Yaskawa INFORM job: X2_NOWY2.JBI

/JOB
//NAME X2_NOWY2
//POS
///NPOS 322,322,322,20,0,0
///TOOL 0
///POSTYPE PULSE
///PULSE
C00000=1579,-114561,-88072,141,60969,-160
C00001=1579,-126069,-115869,130,72161,-147
C00002=-67532,-124352,-115339,134,72718,-152
C00003=-81630,-76415,-67707,7081,99866,-75616
C00004=-81630,-76414,-67706,7081,99866,-75616
C00005=-85213,-86895,-71424,6566,97096,-77009
C00006=-85213,-86471,-70205,6561,96571,-77039
C00007=-85213,-86895,-71424,6566,97096,-77009
C00008=-86383,-83236,-69405,6430,97828,-77376
C00009=-86383,-82993,-68650,6424,97491,-77394
C00010=-85656,-85286,-69628,6508,96860,-77177
C00011=-86054,-83030,-69774,6481,98134,-77248
C00012=-91609,-64546,-67425,5952,106567,-78770
C00013=-108338,-72557,-69392,19017,102016,-84323
C00014=-103994,-87799,-70649,19047,94316,-83966
C00015=-101914,-94753,-72721,19202,91650,-83636
C00016=-101720,-95093,-71454,19192,90702,-83718
C00017=-101720,-95403,-72147,19196,90955,-83679
C00018=-102509,-90897,-70406,19144,92318,-83747
C00019=-102509,-90529,-69509,19136,91974,-83801
C00020=-102070,-93055,-70499,19166,91217,-83763
C00021=-103193,-87364,-70534,19135,94271,-83684
C00022=-105000,-74500,-64879,19101,97659,-83800
C00023=-113069,-60767,-53247,26239,106025,-84622
C00024=-112828,-63942,-52646,27281,108527,-83919
C00025=-112433,-69525,-54608,27546,108328,-83811
C00026=-112433,-69174,-53580,27467,107925,-83912
C00027=-112433,-68598,-51946,27347,107292,-84070
C00028=-112433,-68839,-52622,27396,107553,-84005
C00029=-112673,-65386,-50917,27452,108279,-83921
C00030=-112744,-64051,-49536,27403,108156,-83979
C00031=-112560,-66748,-50889,27360,107600,-84043
C00032=-112776,-63836,-50109,27476,108578,-83887
C00033=-126682,-57830,-51235,23795,116313,-87772
C00034=-91609,-64546,-67425,5952,106567,-78770
C00035=-73590,-134956,-134527,8565,110042,-72105
C00036=-73590,-134956,-134527,8565,110042,-72105
C00037=-85079,-90579,-82104,6699,101738,-76716
C00038=-105233,-99145,-78854,31145,91869,-85162
C00039=-91621,-98116,-75011,30201,81397,-82609
C00040=-84913,-93599,-68771,30087,77670,-80961
C00041=-84913,-92982,-67436,30137,77231,-81076
C00042=-84913,-93205,-67917,30119,77389,-81035
C00043=-86149,-89803,-66593,30086,78643,-81188
C00044=-86149,-89533,-65979,30106,78434,-81245
C00045=-85360,-91719,-66835,30129,77634,-81148
C00046=-89786,-90500,-68269,30172,80536,-82119
C00047=-91499,-86657,-71640,30020,84676,-81700
C00048=-78974,-84836,-79700,7511,102662,-74517
C00049=-79298,-82189,-71657,7361,99132,-74844
C00050=-79260,-81836,-70076,7347,98342,-74878
C00051=-79260,-81218,-68032,7328,97407,-74935
C00052=-79260,-81362,-68495,7333,97617,-74923
C00053=-80441,-78182,-67079,7204,98482,-75282
C00054=-80441,-78012,-66485,7183,98203,-75298
C00055=-79756,-79865,-67316,7258,97705,-75089
C00056=-80252,-78819,-67734,7202,98493,-75213
C00057=-80252,-80316,-73749,7282,101403,-75042
C00058=-98731,-93358,-79222,4709,99471,-81580
C00059=-98353,-93948,-76089,4728,97224,-81535
C00060=-98128,-94312,-74616,4747,96121,-81500
C00061=-98128,-93684,-73071,4742,95494,-81523
C00062=-98128,-93884,-73558,4744,95690,-81516
C00063=-98894,-90114,-72074,4647,96754,-81739
C00064=-98894,-89854,-71388,4644,96467,-81750
C00065=-98435,-92128,-72291,4703,95830,-81616
C00066=-99279,-88707,-72907,4606,98011,-81825
C00067=-99279,-90964,-80150,4662,101298,-81702
C00068=-83031,-73882,-65637,-17912,114082,-77307
C00069=-85653,-78852,-59840,-26006,111225,-77738
C00070=-86395,-77948,-56111,-25174,109013,-77551
C00071=-86395,-77463,-54950,-25096,108589,-77455
C00072=-86395,-77605,-55287,-25118,108711,-77483
C00073=-87408,-74561,-53917,-25584,109056,-77966
C00074=-87408,-74338,-53367,-25545,108852,-77918
C00075=-86830,-76093,-54163,-25280,108655,-77643
C00076=-86155,-69275,-53538,-25095,111477,-78039
C00077=-82305,-66217,-52035,-23871,113209,-76862
C00078=-98731,-93358,-79222,4709,99471,-81580
C00079=-87850,-130184,-128808,6122,98008,-77863
C00080=-131124,-97291,-82060,5244,66687,-6018
C00081=-125790,2337,-22266,13440,105024,83634
C00082=-119533,36956,22492,13071,94512,84678
C00083=-111606,23469,-6781,11265,89839,86812
C00084=-101835,33271,2869,8999,87620,9257
C00085=-96592,41700,11547,7901,86106,-76285
C00086=-96882,40199,11064,7325,85475,-75794
C00087=-96412,39571,15762,7893,82432,-76460
C00088=-96412,39578,15371,7890,82674,-76445
C00089=-96811,43369,19465,7986,82146,-76612
C00090=-96811,43369,19923,7989,81869,-76630
C00091=-96674,42050,18533,7957,82032,-76574
C00092=-96786,43196,17021,7960,83548,-76515
C00093=-105692,32729,6227,9847,85763,-79345
C00094=-105692,32645,7244,9851,85104,-79396
C00095=-105692,32569,8656,9860,84209,-79465
C00096=-105692,32584,8289,9857,84440,-79447
C00097=-105923,35981,11731,9908,84100,-79551
C00098=-105923,35965,12302,9910,83744,-79578
C00099=-105845,34812,11128,9891,83862,-79544
C00100=-105900,35730,9980,9889,85029,-79471
C00101=-105900,36444,4737,9874,88571,-4241
C00102=-111606,23469,-6781,11265,89839,86812
C00103=-109349,27190,646,10801,86931,87307
C00104=-108816,27234,2830,10703,85564,87368
C00105=-108816,27153,4539,10716,84489,87276
C00106=-108816,27166,4149,10713,84731,87297
C00107=-107956,27551,4528,10540,84587,87578
C00108=-108965,27264,1619,10711,86335,87387
C00109=-111260,52324,24435,15027,98353,88139
C00110=-102462,56667,28820,9286,105586,72437
C00111=-101371,54153,30717,9255,103034,72626
C00112=-101300,53253,30624,9243,102627,72619
C00113=-101300,53374,32279,9201,101680,72548
C00114=-101300,53356,32072,9206,101797,72557
C00115=-100938,48635,26847,9267,102537,72740
C00116=-100773,46580,24617,9295,102831,72821
C00117=-101300,53356,32072,9206,101797,72557
C00118=-102175,52590,31226,9140,102021,72268
C00119=-102630,52208,30804,9106,102134,72116
C00120=-102175,52590,31226,9140,102021,72268
C00121=-99428,22928,-9812,4382,95874,-22555
C00122=-101546,17046,-6787,4678,91283,-23411
C00123=-101546,16945,-5416,4675,90390,-23444
C00124=-101514,16566,-4490,4670,89624,-23462
C00125=-101514,16574,-4727,4671,89774,-23457
C00126=-100341,17475,-3893,2784,89101,-18926
C00127=-101749,19095,-4432,4706,90897,-23492
C00128=-101749,19375,-7041,4715,92641,-23427
C00129=-101749,19375,-7041,4715,92641,-23427
C00130=-102981,33005,7118,6834,98538,-23358
C00131=-102660,29046,5283,6805,97611,-23301
C00132=-102660,29002,6609,6789,96777,-23347
C00133=-102660,29022,5897,6798,97224,-23322
C00134=-102541,27735,4980,6792,97060,-7882
C00135=-102724,29871,7085,6794,96879,-7954
C00136=-102669,29379,3677,6831,98706,-7835
C00137=-102669,30744,-3500,6979,103789,-7548
C00138=-89085,-61640,-68335,6227,95184,-3424
C00139=-129723,10180,-8133,7222,98462,-17027
C00140=-105913,33806,-16630,-33387,116609,-16888
C00141=-114766,23108,-3420,-30164,101829,-15972
C00142=-126000,19507,-6631,-29272,96237,-18805
C00143=-125928,21918,3078,-29245,93808,-18174
C00144=-125928,21960,4203,-29214,93219,-18024
C00145=-125927,21943,3808,-29209,93425,-18075
C00146=-125864,24512,6268,-29206,93280,-18014
C00147=-125884,23639,4506,-29235,93832,-18161
C00148=-125884,23787,-988,-29454,96866,-18937
C00149=-117200,23539,-1226,-29926,99884,-16393
C00150=-117161,21121,72,-29726,98116,-15912
C00151=-117144,20144,1246,-29621,97051,-15628
C00152=-117144,20183,2462,-29564,96414,-15463
C00153=-117144,20179,2362,-29568,96466,-15476
C00154=-117212,24135,6125,-29546,96194,-15431
C00155=-117202,23528,1396,-29761,98470,-16021
C00156=-113126,35471,9950,-29950,100652,-15017
C00157=-113126,35383,12410,-29782,99292,-14657
C00158=-113602,35282,14657,-29641,97872,-14469
C00159=-113602,35350,16056,-29571,97148,-14281
C00160=-113602,35312,15354,-29605,97509,-14375
C00161=-114294,35130,15170,-29602,97286,-14585
C00162=-113391,35371,15415,-29607,97577,-14310
C00163=-113626,42883,17073,-29878,99977,-15031
C00164=-136877,41374,10058,10283,103905,-75706
C00165=-141001,35831,8537,10150,102526,-77247
C00166=-140132,39057,14516,9459,103035,-76976
C00167=-140132,39037,16298,9412,101942,-77061
C00168=-140132,39036,16078,9417,102075,-77051
C00169=-140481,35058,11996,9419,102579,-77132
C00170=-140132,39036,16078,9417,102075,-77051
C00171=-138905,38111,15122,9481,102046,-76624
C00172=-140132,39045,14975,9447,102749,-76998
C00173=-140132,39114,13214,9498,103853,-76912
C00174=-141320,34178,2051,14151,101285,-76947
C00175=-141992,34707,2587,2039,92766,-77188
C00176=-132211,33145,3193,-16145,89780,-75832
C00177=-132211,32650,7255,-16139,87130,-75485
C00178=-132167,33411,9664,-16155,86089,-75333
C00179=-132167,33422,9363,-16153,86272,-75358
C00180=-131910,38524,14575,-16205,85759,-75202
C00181=-131910,38519,15135,-16208,85424,-75158
C00182=-131966,37361,13943,-16196,85547,-75193
C00183=-131929,38195,12263,-16188,86960,-75366
C00184=-122451,32022,5983,-17773,89556,-72453
C00185=-122451,31919,7474,-17768,88630,-72319
C00186=-122451,31881,8388,-17768,88076,-72238
C00187=-122451,31892,8078,-17768,88262,-72265
C00188=-122418,36144,12378,-17773,87829,-72190
C00189=-122418,36134,12899,-17774,87518,-72145
C00190=-122425,35123,11870,-17773,87626,-72164
C00191=-122416,36387,11340,-17773,88560,-72297
C00192=-117284,55611,32116,-20493,96434,-72010
C00193=-119259,62166,42313,-20409,96733,-72766
C00194=-130801,68405,49291,-20809,94296,-76538
C00195=-126360,65075,49817,-31825,91468,-75810
C00196=-125594,43121,21590,-30980,86789,-74177
C00197=-141320,33353,7524,13959,97601,-77374
C00198=-139853,30861,8005,10213,95427,-68773
C00199=-139850,30231,7379,10216,95489,-68766
C00200=-141726,26843,4526,13791,96694,-77632
C00201=-141207,31872,9522,12754,100191,-77170
C00202=-131838,40307,17400,-3069,104254,-75449
C00203=-120717,39791,20254,-22002,103322,-74072
C00204=-123241,41817,22993,-23858,102713,-75145
C00205=-120965,41759,25023,-29185,101758,-74907
C00206=-121023,25271,5223,-28433,95326,-73297
C00207=-120372,33506,8504,-28624,97501,-73589
C00208=-120372,33506,8504,-28624,97501,-7388
C00209=-114011,28987,3831,-29482,105348,-6966
C00210=-127301,22883,-362,-9290,98378,-8800
C00211=-130383,22892,110,-12210,96784,-9925
C00212=-119117,21486,5591,-32037,93907,-6966
C00213=-117872,21036,1539,-32238,96305,-7157
C00214=-135561,25772,-1454,-7801,99682,-11540
C00215=-135461,26025,2407,-7746,97466,-11367
C00216=-129197,23357,2778,-20865,94605,-10044
C00217=-129563,23522,5318,-26932,92135,-10188
C00218=-126533,22338,1333,-27220,94758,-9659
C00219=-115633,44815,18495,-18996,108364,22675
C00220=-114107,50921,32807,-24786,104055,23590
C00221=-114339,60935,44009,-24609,102392,23859
C00222=-113327,59043,39697,-24681,104230,23854
C00223=-113549,43239,22387,-25049,106471,23276
C00224=-113959,36250,17368,-26116,100180,17331
C00225=-113750,32141,13338,-26671,97959,14884
C00226=-113784,32033,10394,-26825,99526,14508
C00227=-112924,58292,37776,-24734,105077,23825
C00228=-109456,25709,2980,-23794,97137,26657
C00229=-118237,30699,-4511,6400,110959,24971
C00230=-106534,-87247,-110627,560,89262,27492
C00231=-106534,-87247,-110627,560,89262,27492
C00232=-103790,-60662,-71601,3492,92371,24893
C00233=-90072,-46297,-51679,19403,82444,29914
C00234=-89225,-25796,-38496,19051,95364,28629
C00235=-82968,-19569,-33829,18693,94249,30668
C00236=-92316,-28208,-34631,31848,87681,26801
C00237=-93212,-29211,-40642,31971,90742,27310
C00238=-74629,-7827,-31935,11254,101997,33705
C00239=-71338,-2997,-23236,6798,101883,34323
C00240=-78936,-14568,-30649,16904,94877,32031
C00241=-82428,-18766,-28557,29607,85533,29992
C00242=-85091,-23046,-35219,29948,88128,29642
C00243=-83302,-13788,-26964,29706,87219,30090
C00244=-84406,-14503,-30600,29861,89239,30192
C00245=-85356,-5858,-28119,20956,91780,-33865
C00246=-81588,1907,-17110,16920,91332,-34481
C00247=-80085,-4136,-22119,16745,91007,-34003
C00248=-79500,-6857,-23987,16670,90650,-33848
C00249=-76840,-15565,-30031,18766,92661,-32418
C00250=-81974,-12051,-30981,19262,96095,-33689
C00251=-98247,-31422,-44950,19682,96659,-36405
C00252=-99061,-15599,-30151,19673,95928,-36812
C00253=-99538,-15893,-30372,19693,96028,-36966
C00254=-99542,-11936,-27145,19696,96073,-36959
C00255=-98485,-19802,-33057,19630,95442,-36687
C00256=-97436,-32531,-42916,18662,91677,-32211
C00257=-95696,-34091,-42802,18103,89563,-30497
C00258=-96230,-30895,-40673,18159,89998,-30622
C00259=-92776,-41331,-47434,14269,83214,-21666
C00260=-93749,-43799,-52657,14401,85273,-21763
C00261=-91043,-39779,-53377,13904,87247,-20611
C00262=-86158,-7385,-30463,15366,102993,-69398
C00263=-78323,6041,-20316,6463,111515,-89101
C00264=-75958,-7074,-26718,1279,101463,-89171
C00265=-73720,-14383,-32408,1291,101175,-88413
C00266=-73707,-14423,-32438,1291,101173,-88409
C00267=-74501,-16417,-33720,1350,100398,-77182
C00268=-81364,-12014,-29075,8477,103574,-60369
C00269=-76974,-6126,-24441,8683,103288,-58863
C00270=-85840,-5383,-30241,8443,108111,-61612
C00271=-89409,13061,-14467,8223,108236,-62856
C00272=-89162,11063,-11369,8091,105308,-62973
C00273=-76769,28758,4889,8686,103142,-58806
C00274=-81789,20530,-742,18528,97229,-60276
C00275=-83486,19402,-4941,18704,99513,-60525
C00276=-85618,-23129,-54211,-23,98050,-63088
C00277=-77730,-75302,-67065,7588,99691,-74263
C00278=-69151,-69075,-61356,2748,102855,-72431
C00279=-83665,-83301,-67253,-4133,101740,-77499
C00280=-86539,-83593,-63455,-15981,104296,-78484
C00281=-79657,-74315,-62077,-14413,109372,-76594
C00282=-66263,-128090,-130023,-6185,104579,-72041
C00283=-66263,-128090,-130023,-6185,104579,-72041
C00284=-94568,-90015,-76427,-6942,102962,-81955
C00285=-117694,-91652,-70549,-18356,97186,-89481
C00286=-121556,-93677,-69003,-18900,94414,-90437
C00287=-119795,-72901,-51086,-33493,103547,-78772
C00288=-123287,-66660,-41479,-44294,102063,-75181
C00289=-126428,-64743,-39967,-46087,101055,-75467
C00290=-114717,-64735,-41398,-43474,107786,-72608
C00291=-113328,-78138,-63059,-20614,107376,-72751
C00292=-119993,-75613,-65373,5567,107998,-75141
C00293=-119603,-81287,-64736,5576,104679,-75150
C00294=-101370,-77631,-63119,10020,103783,-68711
C00295=-106562,-79080,-62094,18313,101193,-71017
C00296=-114949,-81063,-65452,19014,103658,-73736
C00297=-107597,-133050,-132520,1199,109480,-70827
C00298=-107600,-133050,-132519,1199,109480,-70827
C00299=-111097,-94755,-74427,15472,95771,-72593
C00300=-108632,-91770,-69991,15763,94145,-71928
C00301=-108459,-93087,-70104,15770,93528,-71947
C00302=-101455,-63232,-52249,14921,110925,-65875
C00303=-99527,-62531,-51785,15542,110635,-65180
C00304=-84477,-49473,-36443,19549,104772,-60394
C00305=-90447,-49925,-33049,29057,101373,-63744
C00306=-112557,-58696,-37857,22594,106874,-71080
C00307=-110623,-74300,-66049,9174,91324,-69507
C00308=-118006,-113386,-124466,9637,107827,-70792
C00309=-118006,-113386,-124466,9637,107827,-70792
C00310=-104411,-100441,-71960,6543,87095,-88178
C00311=-107941,-81766,-58106,7790,96867,-88905
C00312=-111550,-78804,-53150,-16968,99219,-90611
C00313=-100177,-101375,-72775,-10447,90542,-85701
C00314=-127322,-146784,-131564,384,102103,-77635
C00315=-127322,-146784,-131564,384,102103,-77635
C00316=-128319,-94478,-68279,1284,89952,-74935
C00317=-126096,-86443,-60445,1108,95278,-74106
C00318=-113746,-89087,-60975,11490,91598,-70278
C00319=-128822,-103835,-77575,9498,91788,-75427
C00320=-146076,-192209,-136001,7129,84184,-81740
C00321=-146076,-192209,-136001,7129,84184,-81740
BC00000=127053,672594,1075229
BC00001=127053,672594,1075229
BC00002=210750,818892,1075229
BC00003=210750,818892,1005167
BC00004=210749,818892,1005164
BC00005=210749,818892,1005161
BC00006=210749,818892,1005161
BC00007=210749,818892,1005161
BC00008=210749,818892,1005161
BC00009=210749,818892,1005161
BC00010=210749,818892,1005161
BC00011=210749,818892,1005161
BC00012=210749,818892,1005161
BC00013=255741,818892,1005161
BC00014=255741,818892,1005161
BC00015=255741,818892,1005159
BC00016=255741,818892,1005161
BC00017=255741,818892,1005161
BC00018=255741,818892,1005161
BC00019=255741,818892,1005161
BC00020=255741,818892,1005161
BC00021=255741,818892,1005161
BC00022=255741,818892,1005161
BC00023=287623,818892,1005161
BC00024=287623,818892,1005161
BC00025=287623,818892,1005161
BC00026=287623,818892,1005161
BC00027=287623,818892,1005161
BC00028=287623,818892,1005161
BC00029=287623,818892,1005161
BC00030=287623,818892,1005161
BC00031=287623,818892,1005161
BC00032=287623,818892,1005161
BC00033=287623,818892,1005161
BC00034=210749,818892,1005161
BC00035=210749,818892,1005161
BC00036=119260,818892,1005161
BC00037=119260,818892,1005161
BC00038=119260,818892,1005161
BC00039=119260,818892,1005161
BC00040=119260,818892,1005161
BC00041=119260,818892,1005161
BC00042=119260,818892,1005161
BC00043=119260,818892,1005161
BC00044=119260,818892,1005161
BC00045=119260,818892,1005161
BC00046=119260,818892,1005161
BC00047=119260,818892,1005161
BC00048=119260,818892,1005157
BC00049=119260,818892,1005157
BC00050=119260,818892,1005157
BC00051=119260,818892,1005157
BC00052=119260,818892,1005157
BC00053=119260,818892,1005157
BC00054=119261,818892,1005156
BC00055=119261,818892,1005156
BC00056=119260,818892,1005157
BC00057=119260,818892,1005157
BC00058=119260,818892,1005157
BC00059=119260,818892,1005157
BC00060=119260,818892,1005157
BC00061=119260,818892,1005157
BC00062=119260,818892,1005157
BC00063=119260,818892,1005157
BC00064=119260,818892,1005157
BC00065=119260,818892,1005157
BC00066=119260,818892,1005157
BC00067=119260,818892,1005157
BC00068=119260,818892,1005157
BC00069=119260,818892,1005157
BC00070=119260,818892,1005157
BC00071=119260,818892,1005157
BC00072=119260,818892,1005157
BC00073=119260,818892,1005157
BC00074=119260,818892,1005157
BC00075=119260,818892,1005157
BC00076=119260,818892,1005157
BC00077=119260,818892,1005157
BC00078=119260,818892,1005157
BC00079=119260,818892,1005157
BC00080=271066,672595,967916
BC00081=271066,672595,967916
BC00082=271066,672595,967916
BC00083=271066,672595,742596
BC00084=271066,672597,742588
BC00085=271066,672597,742588
BC00086=271066,672597,742588
BC00087=271066,672597,742586
BC00088=271066,672597,742586
BC00089=271066,672597,742586
BC00090=271066,672597,742586
BC00091=271066,672597,742586
BC00092=271066,672597,742586
BC00093=271066,672597,742586
BC00094=271066,672597,742586
BC00095=271066,672597,742586
BC00096=271066,672597,742586
BC00097=271066,672597,742586
BC00098=271066,672597,742586
BC00099=271066,672597,742586
BC00100=271066,672597,742586
BC00101=271066,672597,742586
BC00102=271066,672595,742596
BC00103=271066,672596,742593
BC00104=271066,672596,742593
BC00105=271065,672596,742589
BC00106=271065,672596,742589
BC00107=271065,672596,742589
BC00108=271065,672597,742586
BC00109=271065,672597,742586
BC00110=271065,673087,742586
BC00111=271065,673087,742586
BC00112=271065,673087,742586
BC00113=271065,673087,742586
BC00114=271065,673087,742586
BC00115=271065,673087,742586
BC00116=271065,673087,742586
BC00117=271065,673087,742586
BC00118=271065,673087,742586
BC00119=271065,673087,742586
BC00120=271065,673087,742586
BC00121=271065,673085,742583
BC00122=271065,673085,742583
BC00123=271065,673085,742583
BC00124=271065,673085,742583
BC00125=271065,673085,742583
BC00126=271065,673085,742583
BC00127=271065,673085,742583
BC00128=271065,673085,742583
BC00129=291623,673085,742583
BC00130=291623,673085,742583
BC00131=291623,673085,742583
BC00132=291623,673085,742583
BC00133=291623,673085,742583
BC00134=291623,673085,742583
BC00135=291623,673085,742583
BC00136=291623,673085,742583
BC00137=291623,673085,1054355
BC00138=130801,673085,1059449
BC00139=130802,673083,1031676
BC00140=130802,673083,742569
BC00141=130802,673083,742569
BC00142=130802,673083,742569
BC00143=130802,673083,742569
BC00144=130802,673083,742569
BC00145=130802,673083,742566
BC00146=130802,673083,742566
BC00147=130802,673083,742566
BC00148=130802,673083,742566
BC00149=130802,673083,742566
BC00150=130802,673083,742566
BC00151=130802,673083,742566
BC00152=130802,673083,742566
BC00153=130802,673083,742566
BC00154=130802,673083,742566
BC00155=130802,673083,742566
BC00156=130802,673083,742566
BC00157=130802,673083,742566
BC00158=130802,673083,742566
BC00159=130802,673083,742566
BC00160=130802,673083,742566
BC00161=130802,673083,742566
BC00162=130802,673083,742566
BC00163=130802,673083,742566
BC00164=130802,673083,742566
BC00165=130802,673083,742566
BC00166=130802,673083,742566
BC00167=130802,673083,742566
BC00168=130802,673083,742566
BC00169=130802,673083,742566
BC00170=130802,673083,742566
BC00171=130802,673083,742566
BC00172=130802,673083,742566
BC00173=130802,673083,742566
BC00174=130802,673083,742566
BC00175=130802,673083,742566
BC00176=130802,673083,742566
BC00177=130802,673083,742566
BC00178=130802,673083,742566
BC00179=130802,673083,742566
BC00180=130802,673083,742566
BC00181=130802,673083,742566
BC00182=130802,673083,742566
BC00183=130802,673083,742566
BC00184=130802,673083,742566
BC00185=130802,673083,742566
BC00186=130802,673083,742566
BC00187=130802,673083,742566
BC00188=130802,673083,742566
BC00189=130802,673083,742566
BC00190=130802,673083,742566
BC00191=130802,673083,742566
BC00192=130802,673083,742566
BC00193=130802,673083,742564
BC00194=130802,673083,742560
BC00195=130802,673083,742566
BC00196=130802,673083,742566
BC00197=130802,673083,742566
BC00198=130802,673083,742566
BC00199=130802,673083,742566
BC00200=130802,673083,742566
BC00201=130802,673083,742566
BC00202=130802,673083,742566
BC00203=130802,673083,742566
BC00204=130802,673083,742566
BC00205=130802,673083,742566
BC00206=130802,673083,742566
BC00207=130802,673083,742566
BC00208=130802,673083,742566
BC00209=130802,673083,742566
BC00210=130802,673083,742566
BC00211=130802,673083,742566
BC00212=130802,673083,742566
BC00213=130802,673083,742566
BC00214=130802,673083,742566
BC00215=130802,673083,742566
BC00216=130802,673083,742566
BC00217=130802,673083,742566
BC00218=130802,673083,742566
BC00219=130802,673083,742566
BC00220=130802,673083,742566
BC00221=130802,673083,742566
BC00222=130802,673083,742566
BC00223=130802,673083,742566
BC00224=130802,673083,742566
BC00225=130802,673083,742566
BC00226=130802,673083,742566
BC00227=130802,673083,742566
BC00228=130802,673083,742566
BC00229=130802,673083,742566
BC00230=130802,673083,742566
BC00231=239197,673083,742566
BC00232=239197,748715,742566
BC00233=239197,748715,742566
BC00234=239196,748714,742562
BC00235=239196,748714,742562
BC00236=239196,748714,742562
BC00237=239196,748714,742562
BC00238=239196,748714,742562
BC00239=239196,748714,742562
BC00240=239196,748714,742562
BC00241=239196,748714,742562
BC00242=239196,748714,742562
BC00243=239196,748714,742562
BC00244=239196,748714,742559
BC00245=239196,748714,742559
BC00246=239196,748714,742559
BC00247=239196,748714,742559
BC00248=239196,748714,742559
BC00249=239196,748714,742559
BC00250=239196,748714,742559
BC00251=239196,748714,742559
BC00252=239196,748714,742559
BC00253=239196,748714,742559
BC00254=239196,748714,742559
BC00255=239196,748714,742559
BC00256=239196,748714,742559
BC00257=239196,748714,742559
BC00258=239196,748714,742559
BC00259=239196,748714,742559
BC00260=239196,748714,742559
BC00261=239196,748714,742559
BC00262=239196,748714,742559
BC00263=239196,748714,742559
BC00264=239196,748714,742559
BC00265=239196,748714,742559
BC00266=239196,748714,742559
BC00267=239196,748714,742559
BC00268=239196,748714,742559
BC00269=239196,748714,742559
BC00270=239196,748714,742559
BC00271=239196,748714,742559
BC00272=239196,748714,742559
BC00273=239196,748715,742555
BC00274=239196,748715,742555
BC00275=239196,748715,742555
BC00276=239196,748714,742556
BC00277=210749,818892,1005161
BC00278=210749,818892,1005161
BC00279=210750,818891,1005159
BC00280=210750,818891,1005159
BC00281=210750,818891,1005159
BC00282=210750,818891,1005157
BC00283=123072,818891,1005157
BC00284=123072,818891,1005157
BC00285=162220,818891,1005157
BC00286=162220,818891,1005149
BC00287=162220,818891,1005153
BC00288=162220,818891,1005153
BC00289=162220,818891,1005153
BC00290=162220,818891,1005153
BC00291=162220,818891,1005153
BC00292=162220,818891,1005153
BC00293=162220,818891,1005152
BC00294=162220,818891,1005153
BC00295=162220,818891,1005153
BC00296=162220,818891,1005153
BC00297=162220,818891,1005153
BC00298=264269,818892,1005150
BC00299=264269,818892,1005150
BC00300=264269,818892,1005150
BC00301=264269,818892,1005148
BC00302=264269,818892,1005148
BC00303=264269,818892,1005148
BC00304=264269,818892,1057599
BC00305=264269,818892,1057598
BC00306=264269,818892,1057599
BC00307=264269,818892,1005148
BC00308=264269,818892,1005148
BC00309=150431,818892,1056877
BC00310=150431,818892,1056877
BC00311=150431,818892,1056877
BC00312=150431,818892,1056877
BC00313=150431,818892,1056877
BC00314=150431,818892,1056877
BC00315=276083,818892,1056877
BC00316=276083,818892,1056877
BC00317=276083,818892,1056877
BC00318=276083,818892,1056877
BC00319=276083,818892,1056877
BC00320=276083,818892,1056877
BC00321=276083,684480,1056877
EC00000=-1527674,557300
EC00001=-1527674,557300
EC00002=-1527674,557300
EC00003=-1527674,557300
EC00004=-1527674,557300
EC00005=-1527674,557301
EC00006=-1527674,557301
EC00007=-1527674,557301
EC00008=-1527674,557301
EC00009=-1527674,557301
EC00010=-1527674,557301
EC00011=-1527674,557301
EC00012=-1527674,557301
EC00013=-1527674,557301
EC00014=-1527674,557301
EC00015=-1527674,557301
EC00016=-1527674,557301
EC00017=-1527674,557301
EC00018=-1527674,557301
EC00019=-1527674,557301
EC00020=-1527674,557301
EC00021=-1527674,557301
EC00022=-1527674,557301
EC00023=-1527674,557301
EC00024=-1527674,557301
EC00025=-1527674,557301
EC00026=-1527674,557301
EC00027=-1527674,557301
EC00028=-1527674,557301
EC00029=-1527674,557301
EC00030=-1527674,557301
EC00031=-1527674,557301
EC00032=-1527674,557301
EC00033=-1527674,557301
EC00034=-1527674,557301
EC00035=-1527674,557301
EC00036=-1527674,557301
EC00037=-1527674,557301
EC00038=-1527674,557301
EC00039=-1527674,557301
EC00040=-1527674,557301
EC00041=-1527674,557301
EC00042=-1527674,557301
EC00043=-1527674,557301
EC00044=-1527674,557301
EC00045=-1527674,557301
EC00046=-1527674,557301
EC00047=-1527674,557301
EC00048=-1527675,557301
EC00049=-1527675,557301
EC00050=-1527675,557301
EC00051=-1527675,557301
EC00052=-1527675,557301
EC00053=-1527675,557301
EC00054=-1527675,557301
EC00055=-1527675,557301
EC00056=-1527675,557301
EC00057=-1527675,557301
EC00058=-1527675,557301
EC00059=-1527675,557301
EC00060=-1527675,557301
EC00061=-1527675,557301
EC00062=-1527675,557301
EC00063=-1527675,557301
EC00064=-1527675,557301
EC00065=-1527675,557301
EC00066=-1527675,557301
EC00067=-1527675,557301
EC00068=-1527675,557301
EC00069=-1527675,557301
EC00070=-1527675,557301
EC00071=-1527675,557301
EC00072=-1527675,557301
EC00073=-1527675,557301
EC00074=-1527675,557301
EC00075=-1527675,557301
EC00076=-1527675,557301
EC00077=-1527675,557301
EC00078=-1527675,557301
EC00079=-1527675,557301
EC00080=-1332361,557301
EC00081=-1332361,557301
EC00082=-1332361,557301
EC00083=-1332361,557301
EC00084=-1332360,557303
EC00085=-1332360,557303
EC00086=-1332360,557303
EC00087=-1332360,557303
EC00088=-1332360,557303
EC00089=-1332360,557303
EC00090=-1332360,557303
EC00091=-1332360,557303
EC00092=-1332360,557303
EC00093=-1332360,557303
EC00094=-1332360,557303
EC00095=-1332360,557303
EC00096=-1332360,557303
EC00097=-1332360,557303
EC00098=-1332360,557303
EC00099=-1332360,557303
EC00100=-1332360,557303
EC00101=-1332360,557303
EC00102=-1332361,557301
EC00103=-1332361,557302
EC00104=-1332361,557302
EC00105=-1332361,557302
EC00106=-1332361,557302
EC00107=-1332361,557302
EC00108=-1332361,557302
EC00109=-1332361,557302
EC00110=-1332361,557302
EC00111=-1332361,557302
EC00112=-1332361,557302
EC00113=-1332361,557302
EC00114=-1332361,557302
EC00115=-1332361,557302
EC00116=-1332361,557302
EC00117=-1332361,557302
EC00118=-1332361,557302
EC00119=-1332361,557302
EC00120=-1332361,557302
EC00121=-1332361,557302
EC00122=-1332361,557302
EC00123=-1332361,557302
EC00124=-1332361,557302
EC00125=-1332361,557302
EC00126=-1332361,557302
EC00127=-1332361,557302
EC00128=-1332361,557302
EC00129=-1332361,557302
EC00130=-1332361,557302
EC00131=-1332361,557302
EC00132=-1332361,557302
EC00133=-1332361,557302
EC00134=-1332361,557302
EC00135=-1332361,557302
EC00136=-1332361,557302
EC00137=-1332361,557302
EC00138=-1332361,557302
EC00139=-1332361,557303
EC00140=-1332361,557303
EC00141=-1332361,557303
EC00142=-1332361,557303
EC00143=-1332361,557303
EC00144=-1332361,557303
EC00145=-1332361,557303
EC00146=-1332361,557303
EC00147=-1332361,557303
EC00148=-1332361,557303
EC00149=-1332361,557303
EC00150=-1332361,557303
EC00151=-1332361,557303
EC00152=-1332361,557303
EC00153=-1332361,557303
EC00154=-1332361,557303
EC00155=-1332361,557303
EC00156=-1332361,557303
EC00157=-1332361,557303
EC00158=-1332361,557303
EC00159=-1332361,557303
EC00160=-1332361,557303
EC00161=-1332361,557303
EC00162=-1332361,557303
EC00163=-1332361,557303
EC00164=-1332361,557303
EC00165=-1332361,557303
EC00166=-1332361,557303
EC00167=-1332361,557303
EC00168=-1332361,557303
EC00169=-1332361,557303
EC00170=-1332361,557303
EC00171=-1332361,557303
EC00172=-1332361,557303
EC00173=-1332361,557303
EC00174=-1332361,557303
EC00175=-1332361,557303
EC00176=-1332361,557303
EC00177=-1332361,557303
EC00178=-1332361,557303
EC00179=-1332361,557303
EC00180=-1332361,557303
EC00181=-1332361,557303
EC00182=-1332361,557303
EC00183=-1332361,557303
EC00184=-1332361,557303
EC00185=-1332361,557303
EC00186=-1332361,557303
EC00187=-1332361,557303
EC00188=-1332361,557303
EC00189=-1332361,557303
EC00190=-1332361,557303
EC00191=-1332361,557303
EC00192=-1332361,557303
EC00193=-1332360,557303
EC00194=-1332361,557303
EC00195=-1332361,557303
EC00196=-1332361,557303
EC00197=-1332361,557303
EC00198=-1332361,557303
EC00199=-1332361,557303
EC00200=-1332361,557303
EC00201=-1332361,557303
EC00202=-1332361,557303
EC00203=-1332361,557303
EC00204=-1332361,557303
EC00205=-1332361,557303
EC00206=-1332361,557303
EC00207=-1332361,557303
EC00208=-1332361,557303
EC00209=-1332361,557303
EC00210=-1332361,557303
EC00211=-1332361,557303
EC00212=-1332361,557303
EC00213=-1332361,557303
EC00214=-1332361,557303
EC00215=-1332361,557303
EC00216=-1332361,557303
EC00217=-1332361,557303
EC00218=-1332361,557303
EC00219=-1332361,557303
EC00220=-1332361,557303
EC00221=-1332361,557303
EC00222=-1332361,557303
EC00223=-1332361,557303
EC00224=-1332361,557303
EC00225=-1332361,557303
EC00226=-1332361,557303
EC00227=-1332361,557303
EC00228=-1332361,557303
EC00229=-1332361,557303
EC00230=-1332361,557303
EC00231=-1332361,557303
EC00232=-1332361,557303
EC00233=-1332361,557303
EC00234=-1332361,557303
EC00235=-1332361,557303
EC00236=-1332361,557303
EC00237=-1332361,557303
EC00238=-1332361,557303
EC00239=-1332361,557303
EC00240=-1332361,557303
EC00241=-1332361,557303
EC00242=-1332361,557303
EC00243=-1332361,557303
EC00244=-1332361,557303
EC00245=-1332361,557303
EC00246=-1332361,557303
EC00247=-1332361,557303
EC00248=-1332361,557303
EC00249=-1332361,557303
EC00250=-1332361,557303
EC00251=-1332361,557303
EC00252=-1332361,557303
EC00253=-1332361,557303
EC00254=-1332361,557303
EC00255=-1332361,557303
EC00256=-1332361,557303
EC00257=-1332361,557303
EC00258=-1332361,557303
EC00259=-1332361,557303
EC00260=-1332361,557303
EC00261=-1332361,557303
EC00262=-1332361,557303
EC00263=-1332361,557303
EC00264=-1332361,557303
EC00265=-1332361,557303
EC00266=-1332361,557303
EC00267=-1332361,557303
EC00268=-1332361,557303
EC00269=-1332361,557303
EC00270=-1332361,557303
EC00271=-1332361,557303
EC00272=-1332361,557303
EC00273=-1332360,557303
EC00274=-1332360,557303
EC00275=-1332360,557303
EC00276=-1332361,557303
EC00277=-1527674,557301
EC00278=-1527674,557301
EC00279=-1527675,557301
EC00280=-1527675,557301
EC00281=-1527675,557301
EC00282=-1527675,557302
EC00283=-1527675,557302
EC00284=-1527675,557302
EC00285=-1527675,557302
EC00286=-1527676,557302
EC00287=-1527676,557302
EC00288=-1527676,557302
EC00289=-1527676,557302
EC00290=-1527676,557302
EC00291=-1527676,557302
EC00292=-1527676,557302
EC00293=-1527676,557302
EC00294=-1527676,557302
EC00295=-1527676,557302
EC00296=-1527676,557302
EC00297=-1527676,557302
EC00298=-1527677,557302
EC00299=-1527677,557302
EC00300=-1527677,557302
EC00301=-1527678,557302
EC00302=-1527678,557302
EC00303=-1527678,557302
EC00304=-1527678,557302
EC00305=-1527679,557302
EC00306=-1527678,557302
EC00307=-1527678,557302
EC00308=-1527678,557302
EC00309=-1527678,557302
EC00310=-1527678,557302
EC00311=-1527678,557302
EC00312=-1527678,557302
EC00313=-1527678,557302
EC00314=-1527678,557302
EC00315=-1527678,557302
EC00316=-1527678,557302
EC00317=-1527678,557302
EC00318=-1527678,557302
EC00319=-1527678,557302
EC00320=-1527678,557302
EC00321=-1527678,557302
///POSTYPE BASE
///RECTAN
///RCONF 0,0,0,0,0,0,0,0,0,0,0,0,0,0,0,0,0,0,0,0,0,0,0,0
P00006=0.222,-3.123,-1.508,0.0000,0.0000,0.0000
P00021=-0.225,-6.128,-0.405,0.0000,0.0000,0.0000
P00022=0.222,-3.123,-1.508,0.0000,0.0000,0.0000
P00023=0.143,-0.036,0.682,0.0000,0.0000,0.0000
P00024=0.145,-0.552,1.326,0.0000,0.0000,0.0000
P00025=-2.003,0.006,0.728,0.0000,0.0000,0.0000
P00026=0.562,-0.002,-0.337,0.0000,0.0000,0.0000
P00027=-0.746,0.015,-9.096,0.0000,0.0000,0.0000
P00031=1.853,-0.001,-1.549,0.0000,0.0000,0.0000
P00032=1.957,0.503,-7.217,0.0000,0.0000,0.0000
///RCONF 0,0,0,0,1,0,0,0,0,0,0,0,0,0,0,0,0,0,0,0,0,0,0,0
P00033=-0.123,0.612,-5.012,0.0000,0.0000,0.0000
///RCONF 0,0,0,0,0,0,0,0,0,0,0,0,0,0,0,0,0,0,0,0,0,0,0,0
P00034=-0.304,0.773,-2.693,0.0000,0.0000,0.0000
P00035=2.817,0.591,-1.622,0.0000,0.0000,0.0000
P00036=-1.108,-0.829,1.850,0.0000,0.0000,0.0000
P00037=0.023,0.937,-2.677,0.0000,0.0000,0.0000
P00038=0.158,-1.133,-1.952,0.0000,0.0000,0.0000
P00050=4.296,-4.501,-0.826,0.0000,0.0000,0.0000
P00051=0.367,3.892,0.009,0.0000,0.0000,0.0000
P00052=0.088,2.832,-0.342,0.0000,0.0000,0.0000
P00053=0.134,6.594,0.107,0.0000,0.0000,0.0000
//INST
///DATE 2025/03/13 10:21
///ATTR SC,RW
///GROUP1 RB1,BS1
///GROUP2 ST1
NOP
'PIERWSZA SEKWENCJA
MOVJ C00000 BC00000 VJ=100.00  +MOVJ EC00000 VJ=100.00
MOVJ C00001 BC00001 VJ=100.00  +MOVJ EC00001 VJ=100.00
MOVJ C00002 BC00002 VJ=100.00  +MOVJ EC00002 VJ=100.00
MOVJ C00003 BC00003 VJ=100.00  +MOVJ EC00003 VJ=100.00
SMOVL C00004 BC00004 V=166.7  +MOVJ EC00004
SMOVL C00005 BC00005 V=166.7  +MOVJ EC00005
SREFP 3 C00006 BC00006  +REFP EC00006
CALL JOB:SEARCH-R1-S13D
SET P021 P006
SFTON3D P021
SMOVL C00007 BC00007 V=166.7  +MOVJ EC00007
SMOVL C00008 BC00008 V=83.3  +MOVJ EC00008
SMOVL C00009 BC00009 V=83.3 PL=0  +MOVJ EC00009
SREFP 3 C00010 BC00010  +REFP EC00010
CALL JOB:SEARCH-R1-S13D
SET P021 P006
SFTON3D P021
SMOVL C00011 BC00011 V=166.7  +MOVJ EC00011
MOVL C00012 BC00012 V=800.0  +MOVJ EC00012 VJ=100.00
SFTOF3D
SMOVL C00013 BC00013 V=1000.0  +MOVJ EC00013
SMOVL C00014 BC00014 V=166.7  +MOVJ EC00014
SMOVL C00015 BC00015 V=166.7  +MOVJ EC00015
SREFP 3 C00016 BC00016  +REFP EC00016
CALL JOB:SEARCH-R1-S13D
SET P022 P006
SFTON3D P022
SMOVL C00017 BC00017 V=166.7  +MOVJ EC00017
SMOVL C00018 BC00018 V=166.7  +MOVJ EC00018
SMOVL C00019 BC00019 V=166.7  +MOVJ EC00019
SREFP 3 C00020 BC00020  +REFP EC00020
CALL JOB:SEARCH-R1-S13D
SET P022 P006
SFTON3D P022
SMOVL C00021 BC00021 V=166.7  +MOVJ EC00021
MOVL C00022 BC00022 V=800.0  +MOVJ EC00022 VJ=100.00
SFTOF3D
SMOVL C00023 BC00023 V=1000.0  +MOVJ EC00023
SMOVL C00024 BC00024 V=800.0  +MOVJ EC00024
SMOVL C00025 BC00025 V=166.7  +MOVJ EC00025
SMOVL C00026 BC00026 V=166.7  +MOVJ EC00026
SREFP 3 C00027 BC00027  +REFP EC00027
CALL JOB:SEARCH-R1-S13D
SET P023 P006
SFTON3D P023
SMOVL C00028 BC00028 V=166.7  +MOVJ EC00028
SMOVL C00029 BC00029 V=166.7  +MOVJ EC00029
SMOVL C00030 BC00030 V=166.7  +MOVJ EC00030
SREFP 3 C00031 BC00031  +REFP EC00031
CALL JOB:SEARCH-R1-S13D
SET P023 P006
SFTON3D P023
SMOVL C00032 BC00032 V=166.7  +MOVJ EC00032
MOVL C00033 BC00033 V=800.0  +MOVJ EC00033 VJ=100.00
SFTOF3D
SMOVL C00034 BC00034 V=800.0  +MOVJ EC00034
MOVJ C00035 BC00035 VJ=100.00  +MOVJ EC00035 VJ=100.00
SMOVL C00036 BC00036 V=1000.0  +MOVJ EC00036
SMOVL C00037 BC00037 V=1000.0  +MOVJ EC00037
SMOVL C00038 BC00038 V=1000.0  +MOVJ EC00038
SMOVL C00039 BC00039 V=166.7  +MOVJ EC00039
SMOVL C00040 BC00040 V=166.7  +MOVJ EC00040
SREFP 3 C00041 BC00041  +REFP EC00041
CALL JOB:SEARCH-R1-S13D
SET P024 P006
SFTON3D P024
SMOVL C00042 BC00042 V=166.7  +MOVJ EC00042
SMOVL C00043 BC00043 V=166.7  +MOVJ EC00043
SMOVL C00044 BC00044 V=166.7  +MOVJ EC00044
SREFP 3 C00045 BC00045  +REFP EC00045
CALL JOB:SEARCH-R1-S13D
SET P024 P006
SFTON3D P024
SMOVL C00046 BC00046 V=166.7  +MOVJ EC00046
MOVL C00047 BC00047 V=800.0  +MOVJ EC00047 VJ=100.00
SMOVL C00048 BC00048 V=1000.0  +MOVJ EC00048
SMOVL C00049 BC00049 V=166.7  +MOVJ EC00049
SMOVL C00050 BC00050 V=166.7  +MOVJ EC00050
SREFP 3 C00051 BC00051  +REFP EC00051
CALL JOB:SEARCH-R1-S13D
SET P025 P006
SFTON3D P025
SMOVL C00052 BC00052 V=166.7  +MOVJ EC00052
SMOVL C00053 BC00053 V=166.7  +MOVJ EC00053
SMOVL C00054 BC00054 V=166.7  +MOVJ EC00054
SREFP 3 C00055 BC00055  +REFP EC00055
CALL JOB:SEARCH-R1-S13D
SET P025 P006
SFTON3D P025
SMOVL C00056 BC00056 V=166.7  +MOVJ EC00056
MOVL C00057 BC00057 V=800.0  +MOVJ EC00057 VJ=100.00
SFTOF3D
SMOVL C00058 BC00058 V=1000.0  +MOVJ EC00058
SMOVL C00059 BC00059 V=166.7  +MOVJ EC00059
SMOVL C00060 BC00060 V=166.7  +MOVJ EC00060
SREFP 3 C00061 BC00061  +REFP EC00061
CALL JOB:SEARCH-R1-S13D
SET P026 P006
SFTON3D P026
SMOVL C00062 BC00062 V=166.7  +MOVJ EC00062
SMOVL C00063 BC00063 V=166.7  +MOVJ EC00063
SMOVL C00064 BC00064 V=166.7  +MOVJ EC00064
SREFP 3 C00065 BC00065  +REFP EC00065
CALL JOB:SEARCH-R1-S13D
SET P026 P006
SFTON3D P026
SMOVL C00066 BC00066 V=166.7  +MOVJ EC00066
MOVL C00067 BC00067 V=800.0  +MOVJ EC00067 VJ=100.00
SFTOF3D
SMOVL C00068 BC00068 V=1000.0  +MOVJ EC00068
SMOVL C00069 BC00069 V=166.7  +MOVJ EC00069
SMOVL C00070 BC00070 V=166.7  +MOVJ EC00070
SREFP 3 C00071 BC00071  +REFP EC00071
CALL JOB:SEARCH-R1-S13D
SET P027 P006
SFTON3D P027
SMOVL C00072 BC00072 V=166.7  +MOVJ EC00072
SMOVL C00073 BC00073 V=166.7  +MOVJ EC00073
SMOVL C00074 BC00074 V=166.7  +MOVJ EC00074
SREFP 3 C00075 BC00075  +REFP EC00075
CALL JOB:SEARCH-R1-S13D
SET P027 P006
SFTON3D P027
SMOVL C00076 BC00076 V=166.7  +MOVJ EC00076
MOVL C00077 BC00077 V=800.0  +MOVJ EC00077 VJ=100.00
SFTOF3D
SMOVL C00078 BC00078 V=1000.0  +MOVJ EC00078
MOVJ C00079 BC00079 VJ=80.00  +MOVJ EC00079 VJ=80.00
'DRUGA SEKWENCJA
MOVJ C00080 BC00080 VJ=100.00  +MOVJ EC00080 VJ=100.00
MOVJ C00081 BC00081 VJ=100.00  +MOVJ EC00081 VJ=100.00
MOVJ C00082 BC00082 VJ=100.00  +MOVJ EC00082 VJ=100.00
SMOVL C00083 BC00083 V=1000.0  +MOVJ EC00083
SMOVL C00084 BC00084 V=333.3  +MOVJ EC00084
SMOVL C00085 BC00085 V=333.3  +MOVJ EC00085
SMOVL C00086 BC00086 V=333.3  +MOVJ EC00086
SREFP 3 C00087 BC00087  +REFP EC00087
CALL JOB:SEARCH-R1-S13D
SET P050 P006
SFTON3D P050
SMOVL C00088 BC00088 V=166.7  +MOVJ EC00088
SMOVL C00089 BC00089 V=166.7  +MOVJ EC00089
SMOVL C00090 BC00090 V=166.7  +MOVJ EC00090
SREFP 3 C00091 BC00091  +REFP EC00091
CALL JOB:SEARCH-R1-S13D
SET P050 P006
SFTON3D P050
SMOVL C00092 BC00092 V=166.7  +MOVJ EC00092
SMOVL C00093 BC00093 V=333.3  +MOVJ EC00093
SFTOF3D
SMOVL C00094 BC00094 V=333.3  +MOVJ EC00094
SREFP 3 C00095 BC00095  +REFP EC00095
CALL JOB:SEARCH-R1-S13D
SET P051 P006
SFTON3D P051
SMOVL C00096 BC00096 V=166.7  +MOVJ EC00096
SMOVL C00097 BC00097 V=166.7  +MOVJ EC00097
SMOVL C00098 BC00098 V=166.7  +MOVJ EC00098
SREFP 3 C00099 BC00099  +REFP EC00099
CALL JOB:SEARCH-R1-S13D
SET P051 P006
SFTON3D P051
SMOVL C00100 BC00100 V=166.7  +MOVJ EC00100
SMOVL C00101 BC00101 V=333.3  +MOVJ EC00101
SMOVL C00102 BC00102 V=333.3  +MOVJ EC00102
SMOVL C00103 BC00103 V=166.7  +MOVJ EC00103
SMOVL C00104 BC00104 V=166.7  +MOVJ EC00104
SREFP 3 C00105 BC00105  +REFP EC00105
CALL JOB:SEARCH-R1-S13D
SET P031 P006
SFTON3D P031
SMOVL C00106 BC00106 V=166.7  +MOVJ EC00106
SREFP 3 C00107 BC00107  +REFP EC00107
CALL JOB:SEARCH-R1-S13D
SET P031 P006
SFTON3D P031
SMOVL C00108 BC00108 V=166.7  +MOVJ EC00108
MOVL C00109 BC00109 V=800.0  +MOVJ EC00109 VJ=100.00
SMOVL C00110 BC00110 V=1000.0  +MOVJ EC00110
SFTOF3D
SMOVL C00111 BC00111 V=166.7  +MOVJ EC00111
SMOVL C00112 BC00112 V=166.7  +MOVJ EC00112
SREFP 3 C00113 BC00113  +REFP EC00113
CALL JOB:SEARCH-R1-S13D
SET P032 P006
SFTON3D P032
SMOVL C00114 BC00114 V=166.7  +MOVJ EC00114
SMOVL C00115 BC00115 V=166.7  +MOVJ EC00115
SREFP 3 C00116 BC00116  +REFP EC00116
CALL JOB:SEARCH-R1-S13D
SET P032 P006
SFTON3D P032
SMOVL C00117 BC00117 V=166.7  +MOVJ EC00117
SMOVL C00118 BC00118 V=166.7  +MOVJ EC00118
SREFP 3 C00119 BC00119  +REFP EC00119
CALL JOB:SEARCH-R1-S13D
SET P032 P006
SFTON3D P032
SMOVL C00120 BC00120 V=166.7  +MOVJ EC00120
MOVL C00121 BC00121 V=800.0  +MOVJ EC00121 VJ=100.00
SFTOF3D
SMOVL C00122 BC00122 V=166.7  +MOVJ EC00122
SMOVL C00123 BC00123 V=166.7  +MOVJ EC00123
SREFP 3 C00124 BC00124  +REFP EC00124
CALL JOB:SEARCH-R1-S13D
SET P033 P006
SFTON3D P033
SMOVL C00125 BC00125 V=166.7  +MOVJ EC00125
SREFP 3 C00126 BC00126  +REFP EC00126
CALL JOB:SEARCH-R1-S13D
SET P033 P006
SFTON3D P033
SMOVL C00127 BC00127 V=166.7  +MOVJ EC00127
MOVL C00128 BC00128 V=800.0  +MOVJ EC00128 VJ=100.00
SFTOF3D
SMOVL C00129 BC00129 V=800.0  +MOVJ EC00129
SMOVL C00130 BC00130 V=166.7  +MOVJ EC00130
SMOVL C00131 BC00131 V=166.7  +MOVJ EC00131
SREFP 3 C00132 BC00132  +REFP EC00132
CALL JOB:SEARCH-R1-S13D
SET P034 P006
SFTON3D P034
SMOVL C00133 BC00133 V=166.7  +MOVJ EC00133
SMOVL C00134 BC00134 V=166.7  +MOVJ EC00134
SREFP 3 C00135 BC00135  +REFP EC00135
CALL JOB:SEARCH-R1-S13D
SET P034 P006
SFTON3D P034
SMOVL C00136 BC00136 V=166.7  +MOVJ EC00136
SFTOF3D
MOVL C00137 BC00137 V=1000.0  +MOVJ EC00137 VJ=100.00
MOVJ C00138 BC00138 VJ=100.00  +MOVJ EC00138 VJ=100.00
SMOVL C00139 BC00139 V=1000.0  +MOVJ EC00139
SMOVL C00140 BC00140 V=1000.0  +MOVJ EC00140
SMOVL C00141 BC00141 V=1000.0  +MOVJ EC00141
SMOVL C00142 BC00142 V=166.7  +MOVJ EC00142
SMOVL C00143 BC00143 V=166.7  +MOVJ EC00143
SREFP 3 C00144 BC00144  +REFP EC00144
CALL JOB:SEARCH-R1-S13D
SET P035 P006
SFTON3D P035
SMOVL C00145 BC00145 V=166.7  +MOVJ EC00145
SREFP 3 C00146 BC00146  +REFP EC00146
CALL JOB:SEARCH-R1-S13D
SET P035 P006
SFTON3D P035
SMOVL C00147 BC00147 V=166.7  +MOVJ EC00147
MOVL C00148 BC00148 V=800.0  +MOVJ EC00148 VJ=100.00
SFTOF3D
SMOVL C00149 BC00149 V=1000.0  +MOVJ EC00149
SMOVL C00150 BC00150 V=166.7  +MOVJ EC00150
SMOVL C00151 BC00151 V=166.7  +MOVJ EC00151
SREFP 3 C00152 BC00152  +REFP EC00152
CALL JOB:SEARCH-R1-S13D
SET P036 P006
SFTON3D P036
SMOVL C00153 BC00153 V=166.7  +MOVJ EC00153
SREFP 3 C00154 BC00154  +REFP EC00154
CALL JOB:SEARCH-R1-S13D
SET P036 P006
SFTON3D P036
SMOVL C00155 BC00155 V=166.7  +MOVJ EC00155
SFTOF3D
MOVL C00156 BC00156 V=800.0  +MOVJ EC00156 VJ=100.00
SMOVL C00157 BC00157 V=166.7  +MOVJ EC00157
SMOVL C00158 BC00158 V=166.7  +MOVJ EC00158
SREFP 3 C00159 BC00159  +REFP EC00159
CALL JOB:SEARCH-R1-S13D
SET P038 P006
SFTON3D P038
SMOVL C00160 BC00160 V=166.7  +MOVJ EC00160
SREFP 3 C00161 BC00161  +REFP EC00161
CALL JOB:SEARCH-R1-S13D
SET P038 P006
SFTON3D P038
SMOVL C00162 BC00162 V=166.7  +MOVJ EC00162
MOVL C00163 BC00163 V=800.0  +MOVJ EC00163 VJ=100.00
SFTOF3D
SMOVL C00164 BC00164 V=1000.0  +MOVJ EC00164
SMOVL C00165 BC00165 V=166.7  +MOVJ EC00165
SMOVL C00166 BC00166 V=166.7  +MOVJ EC00166
SREFP 3 C00167 BC00167  +REFP EC00167
CALL JOB:SEARCH-R1-S13D
SET P037 P006
SFTON3D P037
SMOVL C00168 BC00168 V=166.7  +MOVJ EC00168
SREFP 3 C00169 BC00169  +REFP EC00169
CALL JOB:SEARCH-R1-S13D
SET P037 P006
SFTON3D P037
SMOVL C00170 BC00170 V=166.7  +MOVJ EC00170
SREFP 3 C00171 BC00171  +REFP EC00171
CALL JOB:SEARCH-R1-S13D
SET P037 P006
SMOVL C00172 BC00172 V=166.7  +MOVJ EC00172
MOVL C00173 BC00173 V=800.0  +MOVJ EC00173 VJ=100.00
SFTOF3D
SMOVL C00174 BC00174 V=333.3  +MOVJ EC00174
SMOVL C00175 BC00175 V=333.3  +MOVJ EC00175
SMOVL C00176 BC00176 V=333.3  +MOVJ EC00176
SMOVL C00177 BC00177 V=166.7  +MOVJ EC00177
SREFP 3 C00178 BC00178  +REFP EC00178
CALL JOB:SEARCH-R1-S13D
SET P052 P006
SFTON3D P052
SMOVL C00179 BC00179 V=166.7  +MOVJ EC00179
SMOVL C00180 BC00180 V=166.7  +MOVJ EC00180
SMOVL C00181 BC00181 V=166.7  +MOVJ EC00181
SREFP 3 C00182 BC00182  +REFP EC00182
CALL JOB:SEARCH-R1-S13D
SET P052 P006
SFTON3D P052
SMOVL C00183 BC00183 V=166.7  +MOVJ EC00183
SMOVL C00184 BC00184 V=333.3  +MOVJ EC00184
SMOVL C00185 BC00185 V=166.7  +MOVJ EC00185
SREFP 3 C00186 BC00186  +REFP EC00186
CALL JOB:SEARCH-R1-S13D
SET P053 P006
SFTON3D P053
SMOVL C00187 BC00187 V=166.7  +MOVJ EC00187
SMOVL C00188 BC00188 V=166.7  +MOVJ EC00188
SMOVL C00189 BC00189 V=166.7  +MOVJ EC00189
SREFP 3 C00190 BC00190  +REFP EC00190
CALL JOB:SEARCH-R1-S13D
SET P053 P006
SFTON3D P053
SMOVL C00191 BC00191 V=166.7  +MOVJ EC00191
SMOVL C00192 BC00192 V=166.7  +MOVJ EC00192
SMOVL C00193 BC00193 V=166.7 PL=0  +MOVJ EC00193
MACRO1 MJ#(0) ARGF10
ARCON
SFTON3D P052
SMOVL C00194 BC00194 V=8.3  +MOVJ EC00194
SMOVL C00195 BC00195 V=8.3  +MOVJ EC00195
ARCOF
SMOVL C00196 BC00196 V=166.7  +MOVJ EC00196
SMOVL C00197 BC00197 V=800.0  +MOVJ EC00197
MACRO1 MJ#(0) ARGF14
SFTON3D P037
SMOVL C00198 BC00198 V=166.7 PL=0  +MOVJ EC00198
ARCON
SMOVL C00199 BC00199 V=10.0  +MOVJ EC00199
SMOVL C00200 BC00200 V=10.0  +MOVJ EC00200
SMOVC C00201 BC00201 V=10.0  +MOVJ EC00201
SMOVC C00202 BC00202 V=10.0  +MOVJ EC00202
SMOVC C00203 BC00203 V=10.0  +MOVJ EC00203
SMOVL C00204 BC00204 V=10.0  +MOVJ EC00204
SMOVL C00205 BC00205 V=10.0  +MOVJ EC00205
ARCOF
SMOVL C00206 BC00206 V=166.7  +MOVJ EC00206
SFTOF3D
MOVJ C00207 BC00207 VJ=100.00  +MOVJ EC00207 VJ=100.00
MOVJ C00208 BC00208 VJ=100.00  +MOVJ EC00208 VJ=100.00
MOVJ C00209 BC00209 VJ=100.00  +MOVJ EC00209 VJ=100.00
MACRO1 MJ#(0) ARGF10
SFTON3D P035
SMOVL C00210 BC00210 V=166.7  +MOVJ EC00210
ARCON
SMOVL C00211 BC00211 V=6.7  +MOVJ EC00211
MOVL C00212 BC00212 V=6.7  +MOVJ EC00212 VJ=100.00
ARCOF
SMOVL C00213 BC00213 V=166.7  +MOVJ EC00213
SFTOF3D
SMOVL C00214 BC00214 V=166.7  +MOVJ EC00214
SFTON3D P036
SMOVL C00215 BC00215 V=166.7  +MOVJ EC00215
ARCON
SMOVL C00216 BC00216 V=5.8  +MOVJ EC00216
SMOVL C00217 BC00217 V=5.8  +MOVJ EC00217
ARCOF
SMOVL C00218 BC00218 V=166.7  +MOVJ EC00218
SFTOF3D
SMOVL C00219 BC00219 V=166.7  +MOVJ EC00219
SFTON3D P038
MACRO1 MJ#(0) ARGF14
SMOVL C00220 BC00220 V=166.7  +MOVJ EC00220
ARCON
SWVON WEV#(45)
SMOVL C00221 BC00221 V=10.0  +MOVJ EC00221
ARCOF
SWVOF
SFTOF3D
MOVL C00222 BC00222 V=166.7  +MOVJ EC00222 VJ=80.00
MOVL C00223 BC00223 V=166.7  +MOVJ EC00223 VJ=80.00
SFTON3D P038
MOVL C00224 BC00224 V=166.7  +MOVJ EC00224 VJ=80.00
COMM ARCON
MOVL C00225 BC00225 V=8.3  +MOVJ EC00225 VJ=80.00
ARCOF
MOVL C00226 BC00226 V=166.7  +MOVJ EC00226 VJ=80.00
SMOVL C00227 BC00227 V=166.7  +MOVJ EC00227
SFTOF3D
SMOVL C00228 BC00228 V=666.7  +MOVJ EC00228
SMOVL C00229 BC00229 V=666.7  +MOVJ EC00229
SMOVL C00230 BC00230 V=1000.0  +MOVJ EC00230
SMOVL C00231 BC00231 V=1000.0  +MOVJ EC00231
SMOVL C00232 BC00232 V=1000.0  +MOVJ EC00232
SMOVL C00233 BC00233 V=1000.0  +MOVJ EC00233
MACRO1 MJ#(0) ARGF10
SFTON3D P033
SMOVL C00234 BC00234 V=250.0  +MOVJ EC00234
ARCON
SMOVL C00235 BC00235 V=5.8  +MOVJ EC00235
SMOVL C00236 BC00236 V=5.8  +MOVJ EC00236
ARCOF
SFTOF3D
SMOVL C00237 BC00237 V=166.7  +MOVJ EC00237
SMOVL C00238 BC00238 V=166.7  +MOVJ EC00238
SFTON3D P033
SMOVL C00239 BC00239 V=166.7  +MOVJ EC00239
ARCON
SMOVL C00240 BC00240 V=5.8  +MOVJ EC00240
SMOVL C00241 BC00241 V=5.8  +MOVJ EC00241
ARCOF
SMOVL C00242 BC00242 V=250.0  +MOVJ EC00242
MACRO1 MJ#(0) ARGF6
SMOVL C00243 BC00243 V=250.0  +MOVJ EC00243
ARCON
TIMER T=2.00
ARCOF
MOVJ C00244 BC00244 VJ=100.00  +MOVJ EC00244 VJ=100.00
MOVJ C00245 BC00245 VJ=100.00  +MOVJ EC00245 VJ=100.00
MACRO1 MJ#(0) ARGF9
SMOVL C00246 BC00246 V=250.0  +MOVJ EC00246
ARCON
SMOVL C00247 BC00247 V=7.5  +MOVJ EC00247
ARCOF
SMOVL C00248 BC00248 V=7.5  +MOVJ EC00248
ARCON
SMOVL C00249 BC00249 V=7.5  +MOVJ EC00249
ARCOF
SMOVL C00250 BC00250 V=250.0  +MOVJ EC00250
SMOVL C00251 BC00251 V=250.0  +MOVJ EC00251
SFTON3D P031
SREFP 1 C00252 BC00252  +REFP EC00252
SREFP 2 C00253 BC00253  +REFP EC00253
SMOVL C00254 BC00254 V=166.7  +MOVJ EC00254
ARCON
SWVON WEV#(45)
SMOVL C00255 BC00255 V=10.0  +MOVJ EC00255
ARCOF
SWVOF
SMOVL C00256 BC00256 V=133.3  +MOVJ EC00256
SMOVL C00257 BC00257 V=133.3  +MOVJ EC00257
COMM ARCON
SMOVL C00258 BC00258 V=8.3  +MOVJ EC00258
SMOVL C00259 BC00259 V=8.3  +MOVJ EC00259
ARCOF
SMOVL C00260 BC00260 V=250.0  +MOVJ EC00260
MOVJ C00261 BC00261 VJ=100.00  +MOVJ EC00261 VJ=100.00
SFTOF3D
MOVJ C00262 BC00262 VJ=100.00  +MOVJ EC00262 VJ=100.00
MOVJ C00263 BC00263 VJ=100.00  +MOVJ EC00263 VJ=100.00
SFTON3D P032
SMOVL C00264 BC00264 V=250.0  +MOVJ EC00264
MACRO1 MJ#(0) ARGF14
ARCON
SMOVL C00265 BC00265 V=10.0  +MOVJ EC00265
SMOVC C00266 BC00266 V=10.0  +MOVJ EC00266
SMOVC C00267 BC00267 V=10.0  +MOVJ EC00267
SMOVC C00268 BC00268 V=10.0  +MOVJ EC00268
SMOVL C00269 BC00269 V=8.3  +MOVJ EC00269
ARCOF
SMOVL C00270 BC00270 V=250.0  +MOVJ EC00270
SFTOF3D
SFTON3D P050
SMOVL C00271 BC00271 V=333.3  +MOVJ EC00271
SMOVL C00272 BC00272 V=166.7 PL=0  +MOVJ EC00272
MACRO1 MJ#(0) ARGF10
ARCON
SFTON3D P051
SMOVL C00273 BC00273 V=8.3  +MOVJ EC00273
SMOVL C00274 BC00274 V=8.3  +MOVJ EC00274
ARCOF
SMOVL C00275 BC00275 V=333.3  +MOVJ EC00275
SFTOF3D
SMOVL C00276 BC00276 V=666.7  +MOVJ EC00276
MOVJ C00277 BC00277 VJ=100.00  +MOVJ EC00277 VJ=100.00
SFTON3D P021
SMOVL C00278 BC00278 V=166.7 PL=0  +MOVJ EC00278
ARCON
SMOVL C00279 BC00279 V=11.7  +MOVJ EC00279
SMOVL C00280 BC00280 V=11.7  +MOVJ EC00280
ARCOF
SMOVL C00281 BC00281 V=250.0  +MOVJ EC00281
SFTOF3D
SMOVL C00282 BC00282 V=833.3  +MOVJ EC00282
SMOVL C00283 BC00283 V=833.3  +MOVJ EC00283
SMOVL C00284 BC00284 V=833.3  +MOVJ EC00284
SMOVL C00285 BC00285 V=833.3  +MOVJ EC00285
SFTON3D P027
SMOVL C00286 BC00286 V=166.7 PL=0  +MOVJ EC00286
ARCON
SMOVL C00287 BC00287 V=11.7  +MOVJ EC00287
SMOVL C00288 BC00288 V=11.7  +MOVJ EC00288
SMOVL C00289 BC00289 V=11.7  +MOVJ EC00289
ARCOF
SMOVL C00290 BC00290 V=333.3  +MOVJ EC00290
SFTOF3D
SMOVL C00291 BC00291 V=333.3  +MOVJ EC00291
SMOVL C00292 BC00292 V=333.3  +MOVJ EC00292
SFTON3D P025
SMOVL C00293 BC00293 V=166.7 PL=0  +MOVJ EC00293
ARCON
SFTON3D P024
SMOVL C00294 BC00294 V=11.7  +MOVJ EC00294
SMOVL C00295 BC00295 V=11.7  +MOVJ EC00295
ARCOF
SMOVL C00296 BC00296 V=250.0  +MOVJ EC00296
SMOVL C00297 BC00297 V=833.3  +MOVJ EC00297
SMOVL C00298 BC00298 V=833.3  +MOVJ EC00298
SMOVL C00299 BC00299 V=833.3  +MOVJ EC00299
SMOVL C00300 BC00300 V=333.3  +MOVJ EC00300
SFTON3D P022
SMOVL C00301 BC00301 V=166.7 PL=0  +MOVJ EC00301
ARCON
SMOVL C00302 BC00302 V=11.7  +MOVJ EC00302
SMOVL C00303 BC00303 V=11.7  +MOVJ EC00303
SFTON3D P023
SMOVL C00304 BC00304 V=11.7  +MOVJ EC00304
SMOVL C00305 BC00305 V=11.7  +MOVJ EC00305
ARCOF
SMOVL C00306 BC00306 V=250.0  +MOVJ EC00306
SFTOF3D
MOVJ C00307 BC00307 VJ=100.00  +MOVJ EC00307 VJ=100.00
MOVJ C00308 BC00308 VJ=100.00  +MOVJ EC00308 VJ=100.00
MOVJ C00309 BC00309 VJ=100.00  +MOVJ EC00309 VJ=100.00
MOVJ C00310 BC00310 VJ=100.00  +MOVJ EC00310 VJ=100.00
SFTON3D P025
SMOVL C00311 BC00311 V=166.7 PL=0  +MOVJ EC00311
ARCON
SFTON3D P026
SMOVL C00312 BC00312 V=11.7  +MOVJ EC00312
ARCOF
SMOVL C00313 BC00313 V=800.0  +MOVJ EC00313
SFTOF3D
MOVJ C00314 BC00314 VJ=100.00  +MOVJ EC00314 VJ=100.00
MOVJ C00315 BC00315 VJ=100.00  +MOVJ EC00315 VJ=100.00
MOVJ C00316 BC00316 VJ=100.00  +MOVJ EC00316 VJ=100.00
SFTON3D P021
SMOVL C00317 BC00317 V=166.7 PL=0  +MOVJ EC00317
ARCON
SFTON3D P022
SMOVL C00318 BC00318 V=11.7  +MOVJ EC00318
ARCOF
SFTOF3D
SMOVL C00319 BC00319 V=250.0  +MOVJ EC00319
SMOVL C00320 BC00320 V=833.3  +MOVJ EC00320
SMOVL C00321 BC00321 V=833.3  +MOVJ EC00321
END
